FUNCTION PLC_BOOL_TO_LREAL : LREAL
VAR_INPUT
	in: BOOL;
END_VAR
VAR
END_VAR



IF in THEN 
    PLC_BOOL_TO_LREAL := 1.0;
ELSE 
    PLC_BOOL_TO_LREAL := 0.0;
END_IF;

END_FUNCTION

(* stored: Version 1.1.0.1, ProductVersion 3.1.4022.12
   POU PLC_BOOL_TO_LREAL: Id {ac3bc09b-5f96-416d-9711-877bf55364fa}, SpecialFunc None *)
